FUNCTION_BLOCK C_BINARYWRITER
VAR_INPUT
END_VAR
VAR_OUTPUT
END_VAR
VAR
	_BASESTREAM 	: I_STREAM;
END_VAR

PROPERTY BASE_STREAM : I_STREAM
GET
Base_Stream := _BASESTREAM;
END_GET
END_PROPERTY

METHOD CLOSE : DINT
VAR_INPUT
END_VAR
Close := _BASESTREAM.Close();
_BASESTREAM := 0;
RETURN;
END_METHOD

METHOD NEW : DINT
VAR_INPUT
	STREAM : I_STREAM;
END_VAR
IF STREAM = 0 THEN
	New := 1;
	RETURN;
ELSE
	IF STREAM.IsValid THEN
		_BASESTREAM := STREAM;
		_BASESTREAM.Seek( 0, E_STREAMSEEKTYPE.Origin);
		New := -1;
		RETURN;
	ELSE
		New := 1;
		RETURN;
	END_IF
END_IF
END_METHOD

METHOD WRITE_BOOL : DINT
VAR_INPUT
	in_data : BOOL;
END_VAR
IF _BASESTREAM = 0 THEN
	Write_Bool := 1;
	RETURN;
END_IF

Write_Bool := _BASESTREAM.Write(ADR(in_data), 1);
RETURN;
END_METHOD

METHOD WRITE_BYTES : DINT
VAR_INPUT
	in_data 	: POINTER TO BYTE;
	length		: UDINT;
END_VAR
IF _BASESTREAM = 0 THEN
	Write_Bytes := 1;
	RETURN;
END_IF

Write_Bytes := _BASESTREAM.Write(in_data, length);
RETURN;
END_METHOD

METHOD WRITE_DOUBLE : DINT
VAR_INPUT
	in_data : LREAL;
END_VAR
IF _BASESTREAM = 0 THEN
	Write_Double := 1;
	RETURN;
END_IF

Write_Double := _BASESTREAM.Write(ADR(in_data), 8);
RETURN;
END_METHOD

METHOD WRITE_FLOAT : DINT
VAR_INPUT
	in_data : REAL;
END_VAR
IF _BASESTREAM = 0 THEN
	Write_Float := 1;
	RETURN;
END_IF

Write_Float := _BASESTREAM.Write(ADR(in_data) , 4);
RETURN;
END_METHOD

METHOD WRITE_INT16 : DINT
VAR_INPUT
	in_data : INT;
END_VAR
IF _BASESTREAM = 0 THEN
	Write_Int16 := 1;
	RETURN;
END_IF

Write_Int16 := _BASESTREAM.Write(ADR(in_data) , 2);
RETURN;
END_METHOD

METHOD WRITE_INT32 : DINT
VAR_INPUT
	in_data : DINT;
END_VAR
IF _BASESTREAM = 0 THEN
	Write_Int32 := 1;
	RETURN;
END_IF

Write_Int32 := _BASESTREAM.Write(ADR(in_data) , 4);
RETURN;
END_METHOD

METHOD WRITE_STRING : DINT
VAR_INPUT
	in_data 	: PVOID;
	length		: UDINT;
END_VAR
IF _BASESTREAM = 0 THEN
	Write_String := 1;
	RETURN;
END_IF

Write_String := _BASESTREAM.Write(in_data, length);
RETURN;
END_METHOD

METHOD WRITE_UINT16 : DINT
VAR_INPUT
	in_data : UINT;
END_VAR
IF _BASESTREAM = 0 THEN
	Write_UInt16 := 1;
	RETURN;
END_IF

Write_UInt16 := _BASESTREAM.Write(ADR(in_data) , 4);
RETURN;
END_METHOD

METHOD WRITE_UINT32 : DINT
VAR_INPUT
	in_data : UDINT;
END_VAR
IF _BASESTREAM = 0 THEN
	Write_UInt32 := 1;
	RETURN;
END_IF

Write_UInt32 := _BASESTREAM.Write(ADR(in_data) , 4);
RETURN;
END_METHOD

END_FUNCTION_BLOCK

(* stored: Version 1.1.0.1, ProductVersion 3.1.4020.3
   POU C_BINARYWRITER: Id {e7f30169-cf04-41d2-b79c-23b5695cf795}, SpecialFunc None
   Property BASE_STREAM: Id {3dcd12a4-e306-49ed-938a-5220871db64f}
   Get Get: Id {85b4857b-a5ab-4898-8488-7d4e7f67ebe9}
   Method CLOSE: Id {af4be7ee-df55-43f8-882b-81de066d5a72}
   Method NEW: Id {bf9e58ea-41d9-42ca-a471-045ce927c089}
   Method WRITE_BOOL: Id {7743df79-e2d5-49de-99a2-359a2ae83fbb}
   Method WRITE_BYTES: Id {c5f6e455-1e48-420b-aadf-1ba979cd59eb}
   Method WRITE_DOUBLE: Id {fc137834-c546-4ead-91d9-c3027d0be7cc}
   Method WRITE_FLOAT: Id {8d1e632b-d11a-42b0-8774-953d07c3b7e8}
   Method WRITE_INT16: Id {15bcfc73-e915-4034-a81f-7f040d017fa0}
   Method WRITE_INT32: Id {904892c4-4133-4397-a7df-060fbc4a953e}
   Method WRITE_STRING: Id {7115c34f-7f55-4080-97ae-652a8e87cc88}
   Method WRITE_UINT16: Id {55423954-4581-4831-bdfd-662fd3d0727d}
   Method WRITE_UINT32: Id {6ec8e28c-8c95-4b09-a9e3-dca4cf6121f6} *)
